Universal Robots PolyScope program: SocketTCP_ex_pose.urp

Program interfaces_m3t4 (installation=default directory=/programs/usbdisk createdIn=5.11.1 lastSavedIn=5.13.1 robotSerialNumber=20205500771)
Calibrated DH parameters: a=[0.00017, -0.315777, -0.390584, 0.000089, 0.000022, 0]; d=[0.16289, -151.810109, 155.986099, -4.043122, 0.099816, 0.099706]; alpha=[1.572969, -0.001875, 0.009547, 1.571313, -1.570827, 0]; deltaTheta=[0, 0.733614, -0.631905, -0.101721, 0.000001, 0]
InitVariablesNode
BeforeStart
  'Interfaces Module 3 Task 2'
  'receive pose coordinates to move to from the server'
  conn := False
  counter := 0
  progress := False
Robot Program (runOnlyOnce=true)
  Folder establish connection
    Loop While (checkContinuously=false) expression=conn≟ False
      conn := socket_open("192.168.0.12", 1701, "soc_name")
      Wait Sleep waitTime=2
      counter := counter+1
      progress := True
      Wait Sleep waitTime=5
      str := "ready"
      Script: socket_send_string(str, "soc_name")
      Script: socket_send_byte(13, "soc_name")
      Script: socket_send_byte(10, "soc_name")
  Wait Sleep waitTime=1
  Folder get and send current status
    current_pos := get_actual_tcp_pose()
    current_joints := get_actual_joint_positions()
    Script: socket_send_string("current position is: ", "soc_name")
    str := to_str(current_pos)
    Script: socket_send_string(str, "soc_name")
    Script: socket_send_byte(13, "soc_name")
    Script: socket_send_byte(10, "soc_name")
    Script: socket_send_string("current joint angles in radians is: ", "soc_name")
    str := to_str(current_joints)
    Script: socket_send_string(str, "soc_name")
    Script: socket_send_byte(13, "soc_name")
    Script: socket_send_byte(10, "soc_name")
  Folder ask for the waypoint to move to
    str := "where should the robot move to? format your response in parentheses as (x,y,z,rx,ry,rz): "
    Script: socket_send_string(str, "soc_name")
    Script: socket_send_byte(13, "soc_name")
    Script: socket_send_byte(10, "soc_name")
  Wait Sleep waitTime=1
  Folder read in the waypoint
    num_intake := [0,0,0,0,0,0,0]
    Loop While (checkContinuously=false) expression=num_intake[0]≟0
      num_intake := socket_read_ascii_float(6, "soc_name")
      Wait Sleep waitTime=0.1
    str := "loop variable recieved "
    Script: socket_send_string(str, "soc_name")
    Script: socket_send_byte(13, "soc_name")
    Script: socket_send_byte(10, "soc_name")
    Folder process into waypoint
      target_pos := p[0,0,0,0,0,0]
      Script: target_pos[0]=num_intake[1]
      Script: target_pos[1]=num_intake[2]
      Script: target_pos[2]=num_intake[3]
      Script: target_pos[3]=num_intake[4]
      Script: target_pos[4]=num_intake[5]
      Script: target_pos[5]=num_intake[6]
  Wait Sleep waitTime=1
  Folder move to the waypoint
    MoveJ speed 30 deg/s, acceleration 30 deg/s^2 (useActiveTCP=true) feature=Base
      Waypoint Variable (Variable): variable(name=target_pos)
  Wait Sleep waitTime=5
  Script: socket_close()
